TYPE AbbLinkinRequest_Typ :
STRUCT
	command		: ABBLINKIN_COMMAND_TYPE;
	uri			: STRING;
	httpMethod	: ETcIotHttpRequestType;
	pContent	: PVOID;
	contentSize	: UDINT;
	pStatus		: POINTER TO AbbLinkinRequestStatus_Typ;
	pResults	: POINTER TO AbbLinkinGetterResults_Typ;
END_STRUCT
END_TYPE

(* stored: Version 1.1.0.1, ProductVersion 3.1.4024.12
   DUT AbbLinkinRequest_Typ: Id {9d01c7cf-9f93-4ceb-b209-32052c2214ca} *)
